{attribute 'qualified_only'}
{attribute 'strict'}
TYPE ST_PalletStopHardwareStates :
(
	enum_member := 0
);
END_TYPE

(* stored: Version 1.1.0.1, ProductVersion 3.1.4024.12
   DUT ST_PalletStopHardwareStates: Id {abf2666a-2bd9-497c-aa01-1355d28f81b8} *)
